{attribute addProperty BoxType "EL3483-0000-0016"}
{attribute addProperty Id "System_StateAT %I*BOOL811Grid_DirectionAT %I*BOOL812Frequency_Guard_WarningAT %I*BOOL813Frequency_Guard_ErrorAT %I*BOOL814Power_Quality_Guard_WarningAT %I*BOOL8111Power_Quality_Guard_ErrorAT %I*BOOL8112TxPDO_StateAT %I*BOOL8115TxPDO_ToggleAT %I*BOOL8116Power_Quality_FactorAT %I*REAL32417"}
{attribute addProperty CRC "1382465625"}
{attribute addProperty SizeInBites "96"}
{attribute addProperty SizeInBytes "12"}
TYPE Total_Status_5266C059 :
STRUCT
	{attribute addProperty Name "System_State"}
	System_State AT %I* : BOOL;
	{attribute addProperty Name "Grid_Direction"}
	Grid_Direction AT %I* : BOOL;
	{attribute addProperty Name "Frequency_Guard_Warning"}
	Frequency_Guard_Warning AT %I* : BOOL;
	{attribute addProperty Name "Frequency_Guard_Error"}
	Frequency_Guard_Error AT %I* : BOOL;
	{attribute addProperty Name "Power_Quality_Guard_Warning"}
	Power_Quality_Guard_Warning AT %I* : BOOL;
	{attribute addProperty Name "Power_Quality_Guard_Error"}
	Power_Quality_Guard_Error AT %I* : BOOL;
	{attribute addProperty Name "TxPDO_State"}
	TxPDO_State AT %I* : BOOL;
	{attribute addProperty Name "TxPDO_Toggle"}
	TxPDO_Toggle AT %I* : BOOL;
	{attribute addProperty Name "Power_Quality_Factor"}
	Power_Quality_Factor AT %I* : REAL;
END_STRUCT
END_TYPE

(* stored: Version 1.2.0.0, ProductVersion 3.1.4024.9
   DUT Total_Status_5266C059: Id {ae611060-f7ff-4433-a142-6dc954793cfb} *)
